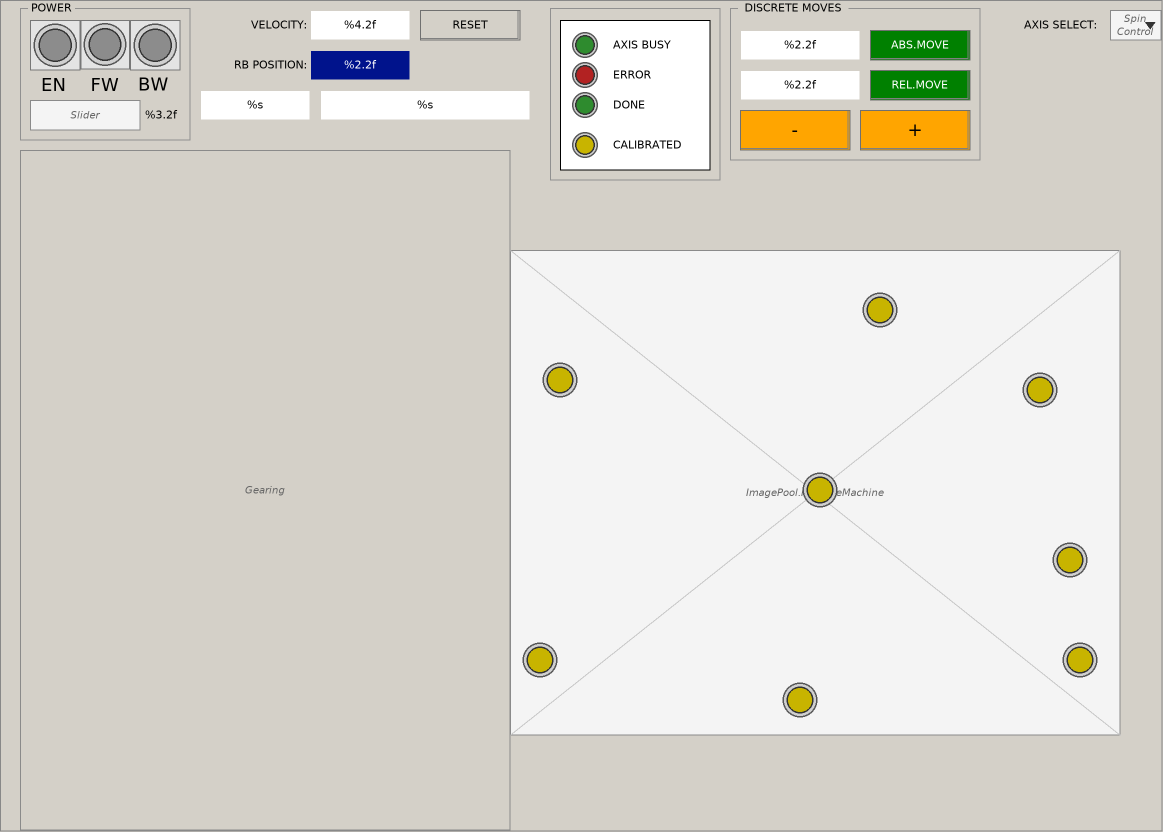
VISUALIZATION Visualization  // 1163x832
    GroupBox (730,0 250x160), "DISCRETE MOVES"
        Textfield (10,30 120x30), "%2.2f", text variable: MAIN.axes[MAIN.hmiAxisSelect].fPosition
            OnMouseClick: write MAIN.axes[MAIN.hmiAxisSelect].fPosition via Default
        Button (140,30 100x30), "ABS.MOVE", input disabled if: MAIN.axes[MAIN.hmiAxisSelect].iAxisState=500
            OnMouseClick: execute { MAIN.axes[MAIN.hmiAxisSelect].eCommand:=McCommand.MoveAbsolute; MAIN.axes[MAIN.hmiAxisSelect].bEXECUTE:= TRUE; }
        Textfield (10,70 120x30), "%2.2f", text variable: MAIN.axes[MAIN.hmiAxisSelect].fDistance
            OnMouseClick: write MAIN.axes[MAIN.hmiAxisSelect].fDistance via Default
        Button (140,70 100x30), "REL.MOVE", input disabled if: MAIN.axes[MAIN.hmiAxisSelect].iAxisState=500
            OnMouseClick: execute { MAIN.axes[MAIN.hmiAxisSelect].eCommand:=McCommand.MoveRelative; MAIN.axes[MAIN.hmiAxisSelect].bEXECUTE:= TRUE; }
        Button (10,110 110x40), "-"
            tap MAIN.axes[MAIN.hmiAxisSelect].bJogBackward
            OnMouseClick: execute { MAIN.axes[MAIN.hmiAxisSelect].eCommand:=McCommand.Jog; }
        Button (130,110 110x40), "+"
            tap MAIN.axes[MAIN.hmiAxisSelect].bJogForward
            OnMouseClick: execute { MAIN.axes[MAIN.hmiAxisSelect].eCommand:=McCommand.Jog; }
    Textfield (310,50 100x30), "%2.2f", text variable: MAIN.axes[MAIN.hmiAxisSelect].Axis.NcToPlc.ActPos
    SpinControl (1110,10 51x30), variable: MAIN.hmiAxisSelect
        p651134158: GVL.axisNumMax
    Textfield (310,10 100x30), "%4.2f", text variable: MAIN.axes[MAIN.hmiAxisSelect].fVelocity
        OnMouseClick: write MAIN.axes[MAIN.hmiAxisSelect].fVelocity via Default
    Textfield (980,10 120x30), "AXIS SELECT:", text variable: MAIN.hmiAxisSelect
    Textfield (190,10 120x30), "VELOCITY:", text variable: MAIN.hmiAxisSelect
    Textfield (190,50 120x30), "RB POSITION:"
    GroupBox (20,0 170x140), "POWER"
        PushSwitchLed (10,20 50x50), variable: MAIN.axes[MAIN.hmiAxisSelect].bEnable, behaviour: TOGGLE, style: Switch-PushSwitchLed-Gray
        PushSwitchLed (110,20 50x50), variable: Limits.BwLimit[MAIN.hmiAxisSelect], behaviour: TOGGLE, style: Switch-PushSwitchLed-Gray
        Slider (10,100 110x30), variable: MAIN.axes[MAIN.hmiAxisSelect].fOverride, scale 0..100
        Textfield (120,100 40x30), "%3.2f", text variable: MAIN.axes[hmiAxisSelect].fOverride
        Label (10,70 47x30), "EN"
        Label (110,70 47x29), "BW"
        PushSwitchLed (60,20 50x49), variable: Limits.FwLimit[MAIN.hmiAxisSelect], behaviour: TOGGLE, style: Switch-PushSwitchLed-Gray
        Label (60,70 50x30), "FW"
    GroupBox (550,0 170x180)
        Rectangle (10,20 150x150)
        Lamp1 (20,30 30x30), variable: MAIN.axes[MAIN.hmiAxisSelect].bBusy, style: Lamp-Lamp1-Green
        Lamp1 (20,60 30x30), variable: MAIN.axes[MAIN.hmiAxisSelect].bError, style: Lamp-Lamp1-Red
        Lamp1 (20,90 30x30), variable: MAIN.axes[MAIN.hmiAxisSelect].bDone, style: Lamp-Lamp1-Green
        Textfield (60,30 90x30), "AXIS BUSY", text variable: MAIN.hmiAxisSelect
        Textfield (60,60 90x30), "ERROR", text variable: MAIN.hmiAxisSelect
        Textfield (60,90 90x30), "DONE", text variable: MAIN.hmiAxisSelect
        Lamp1 (20,130 30x30), variable: MAIN.axes[MAIN.hmiAxisSelect].Axis.Status.Homed, style: Lamp-Lamp1-Yellow
        Textfield (60,130 90x30), "CALIBRATED", text variable: MAIN.hmiAxisSelect
    Textfield (200,90 110x30), "%s", text variable: MAIN.axes[MAIN.hmiAxisSelect].sAxisName
        OnMouseClick: write MAIN.axes[MAIN.hmiAxisSelect].sAxisName via Edit
    Textfield (320,90 210x30), "%s", text variable: MAIN.axes[MAIN.hmiAxisSelect].sAxisDesc
        OnMouseClick: write MAIN.axes[MAIN.hmiAxisSelect].sAxisDesc via Edit
    Button (420,10 100x30), "RESET"
        OnMouseClick: execute { MAIN.axes[MAIN.hmiAxisSelect].eCommand:=McCommand.Reset; MAIN.axes[MAIN.hmiAxisSelect].bReset:= TRUE; }
    Image (510,250 610x485), image: ImagePool.NCStateMachine
    Lamp1 (1060,640 40x40), variable: MAIN.axes[MAIN.hmiAxisSelect].iAxisState=100, style: Lamp-Lamp1-Yellow
    Lamp1 (780,680 40x40), variable: MAIN.axes[MAIN.hmiAxisSelect].iAxisState=200, style: Lamp-Lamp1-Yellow
    Lamp1 (520,640 40x40), variable: MAIN.axes[MAIN.hmiAxisSelect].iAxisState=300, style: Lamp-Lamp1-Yellow
    Lamp1 (1050,540 40x40), variable: MAIN.axes[MAIN.hmiAxisSelect].iAxisState=999, style: Lamp-Lamp1-Yellow
    Lamp1 (800,470 40x40), variable: MAIN.axes[MAIN.hmiAxisSelect].iAxisState=700, style: Lamp-Lamp1-Yellow
    Lamp1 (1020,370 40x40), variable: MAIN.axes[MAIN.hmiAxisSelect].iAxisState=600, style: Lamp-Lamp1-Yellow
    Lamp1 (540,360 40x40), variable: MAIN.axes[MAIN.hmiAxisSelect].iAxisState=400, style: Lamp-Lamp1-Yellow
    Lamp1 (860,290 40x40), variable: MAIN.axes[MAIN.hmiAxisSelect].iAxisState=500, style: Lamp-Lamp1-Yellow
    TabControl (20,150 490x680)
        shows Gearing()
        shows Parameters()
        shows Homing()
        shows AxisSimulation()
        [0]: TabTitle=Gearing
        [1]: TabTitle=Parameters
        [2]: TabTitle=Adv. Homing
        [3]: TabTitle=Simulation
END_VISUALIZATION

(* stored: Version 1.1.0.1, ProductVersion 3.1.4020.12
   Visu Visualization: Id {91dd2de5-17c4-4aa2-8a01-4e0028983367} *)
